PROGRAM Taster_entprellung
VAR
	SR1: SR;
	SR2: SR;
END_VAR

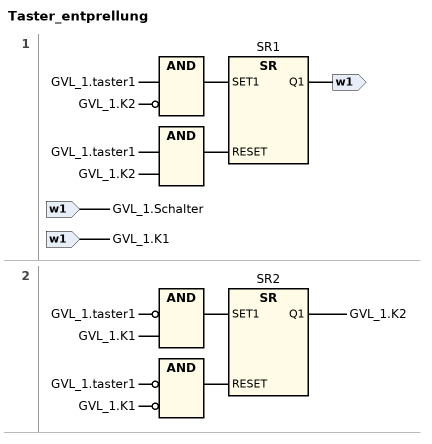
// NETWORK 1
SR1(SET1 := GVL_1.taster1 AND NOT GVL_1.K2, RESET := GVL_1.taster1 AND GVL_1.K2); // SR
GVL_1.Schalter := SR1.Q1;
GVL_1.K1 := SR1.Q1;

// NETWORK 2
SR2(SET1 := NOT GVL_1.taster1 AND GVL_1.K1, RESET := NOT GVL_1.taster1 AND NOT GVL_1.K1); // SR
GVL_1.K2 := SR2.Q1;

END_PROGRAM

(* stored: Version 1.1.0.1, ProductVersion 3.1.4022.9
   POU Taster_entprellung: Id {4a40d1bb-ea83-4bc5-af29-d969329bf5e6}, SpecialFunc None *)
